Yaskawa INFORM job: R2_W24(KAMERA)(-90,90)-OKAW!!.JBI

/JOB
//NAME R2_W24(KAMERA)(-90,90)-OKAW!!
///FOLDERNAME MP_TEST
//POS
///NPOS 54,54,0,5,0,0
///TOOL 0
///POSTYPE PULSE
///PULSE
C00000=123600,-12860,-54312,-41640,88148,80397
C00001=123600,-12860,-54312,-41640,88148,80397
C00002=120727,72264,45486,-43419,68187,78537
C00003=120730,72194,45402,-43416,68199,78533
C00004=120680,125282,114040,-48791,57564,83971
C00005=120680,105365,87155,-46138,61919,81546
C00006=120233,105377,87170,-46014,61686,81428
C00007=120680,105365,87155,-46138,61919,81546
C00008=120680,106282,89568,-46525,61204,81923
C00009=120680,105365,87155,-46138,61919,81546
C00010=120680,105137,86855,-46113,61967,81521
C00011=120680,105137,86855,-46113,61967,81521
C00012=120680,105137,86855,-46113,61967,81521
C00013=120282,105147,86868,-46001,61759,81415
C00014=120680,105137,86855,-46113,61967,81521
C00015=120680,105947,89012,-46459,61327,81858
C00016=120680,105137,86855,-46113,61967,81521
C00017=126632,103319,76893,-46095,68710,81214
C00018=105628,110861,70631,9181,76248,77143
C00019=90079,103598,72277,44137,82752,76276
C00020=94241,81988,53921,45576,81194,77750
C00021=94241,81988,53921,45576,81194,77750
C00022=94870,80971,52672,45434,81052,77981
C00023=94241,81988,53921,45576,81194,77750
C00024=94241,82066,55088,45641,80710,77527
C00025=94241,81988,53921,45576,81194,77750
C00026=90439,80786,48344,46103,85116,77771
C00027=91144,88736,58191,46078,83363,77287
C00028=93989,78186,49515,45558,81861,77938
C00029=93989,78186,49515,45558,81861,77938
C00030=94486,77409,48575,45448,81739,78115
C00031=93989,78186,49515,45558,81861,77938
C00032=93989,78219,50499,45608,81441,77746
C00033=93989,78186,49515,45558,81861,77938
C00034=89014,87596,51414,46328,86969,77970
C00035=117044,71985,11723,-22209,90241,74173
C00036=120735,72113,44062,-43216,68780,78274
C00037=121402,72146,45355,-43635,68530,78708
C00038=124662,56949,12200,-42482,79430,75485
C00039=120367,52960,24213,-42516,70372,77401
C00040=120494,108785,92194,-46600,60881,81998
C00041=120821,102740,83763,-45903,62519,81314
C00042=122365,100198,76797,-45341,65431,80657
C00043=120730,72194,45403,-43416,68199,78533
C00044=107638,83716,21915,3272,91251,77584
C00045=122737,105379,80503,39421,63908,84000
C00046=124412,110163,91084,40204,59985,83172
C00047=120735,72112,44061,-43216,68781,78273
C00048=121402,72146,45354,-43635,68530,78708
C00049=124480,110073,90880,40152,60017,83221
C00050=124522,108531,89026,40010,60267,83350
C00051=123404,106925,84118,39642,62487,83737
C00052=116116,74146,21472,33448,73223,88073
C00053=116116,87806,16032,32344,82007,90677
BC00000=160885,285292,992696
BC00001=160885,285292,992696
BC00002=159740,272384,1010808
BC00003=159782,272389,903274
BC00004=165429,271706,884467
BC00005=165429,264224,884467
BC00006=165429,264224,884467
BC00007=165429,264224,884467
BC00008=165429,264224,884467
BC00009=165429,264224,884467
BC00010=148950,189766,914170
BC00011=165429,189766,884467
BC00012=165429,189766,884467
BC00013=165429,189766,884467
BC00014=165429,189766,884467
BC00015=165429,189766,884467
BC00016=165429,189766,884467
BC00017=165429,189766,884467
BC00018=165429,189766,884467
BC00019=165429,165645,884467
BC00020=165429,165645,884467
BC00021=165429,165645,884467
BC00022=165429,165645,884467
BC00023=165429,165645,884467
BC00024=165429,165645,884467
BC00025=165429,165645,884467
BC00026=165429,165645,884467
BC00027=165429,230278,884467
BC00028=165429,230278,884467
BC00029=165429,230278,884467
BC00030=165429,230278,884467
BC00031=165429,230278,884467
BC00032=165429,230278,884467
BC00033=165429,230278,884467
BC00034=165429,230278,884467
BC00035=166074,230142,881925
BC00036=167687,271433,876944
BC00037=167687,271433,876944
BC00038=166263,230102,881180
BC00039=166263,230102,881180
BC00040=166263,230102,881180
BC00041=167434,171755,876574
BC00042=167434,171755,876574
BC00043=159528,215497,902904
BC00044=167434,242986,876574
BC00045=273098,271706,884467
BC00046=273098,271706,884467
BC00047=167961,332876,877344
BC00048=167961,332876,877344
BC00049=273098,231841,884467
BC00050=273098,175866,884467
BC00051=273098,175866,884467
BC00052=273098,218083,884467
BC00053=273098,304310,884467
///POSTYPE BASE
///RECTAN
///RCONF 0,0,0,0,0,0,0,0,0,0,0,0,0,0,0,0,0,0,0,0,0,0,0,0
P00006=0.222,-3.123,-1.508,0.0000,0.0000,0.0000
P00021=-0.225,-6.128,-0.405,0.0000,0.0000,0.0000
P00022=0.222,-3.123,-1.508,0.0000,0.0000,0.0000
P00023=0.143,-0.036,0.682,0.0000,0.0000,0.0000
P00024=0.145,-0.552,1.326,0.0000,0.0000,0.0000
//INST
///DATE 2023/11/22 15:59
///ATTR SC,RW
///GROUP1 RB1,BS1
NOP
'r2_W24(kamera)(-90,90)
'Path W790
SFTOF
MOVJ C00000 BC00000 VJ=20.00
CALL JOB:CLEAN-R1_LONG
MOVJ C00001 BC00001 VJ=20.00
MOVJ C00002 BC00002 VJ=20.00
MOVJ C00003 BC00003 VJ=20.00
MOVJ C00004 BC00004 VJ=20.00
MOVL C00005 BC00005 V=60.0
REFP 3 C00006 BC00006
CALL JOB:SEARCH-R1
SET P021 P006
SFTON P021
MOVL C00007 BC00007 V=60.0
REFP 3 C00008 BC00008
CALL JOB:SEARCH-R1
SET P021 P006
SFTON P021
MOVL C00009 BC00009 V=60.0
MOVJ C00010 BC00010 VJ=20.00
MOVJ C00011 BC00011 VJ=20.00
MOVL C00012 BC00012 V=60.0
REFP 3 C00013 BC00013
CALL JOB:SEARCH-R1
SET P022 P006
SFTON P022
MOVL C00014 BC00014 V=60.0
REFP 3 C00015 BC00015
CALL JOB:SEARCH-R1
SET P022 P006
SFTON P022
MOVL C00016 BC00016 V=60.0
MOVJ C00017 BC00017 VJ=20.00
MOVJ C00018 BC00018 VJ=20.00
MOVJ C00019 BC00019 VJ=20.00
MOVJ C00020 BC00020 VJ=20.00
MOVL C00021 BC00021 V=60.0
REFP 3 C00022 BC00022
CALL JOB:SEARCH-R1
SET P023 P006
SFTON P023
MOVL C00023 BC00023 V=60.0
REFP 3 C00024 BC00024
CALL JOB:SEARCH-R1
SET P023 P006
SFTON P023
MOVL C00025 BC00025 V=60.0
MOVJ C00026 BC00026 VJ=20.00
MOVJ C00027 BC00027 VJ=20.00
MOVJ C00028 BC00028 VJ=20.00
MOVL C00029 BC00029 V=60.0
REFP 3 C00030 BC00030
CALL JOB:SEARCH-R1
SET P024 P006
SFTON P024
MOVL C00031 BC00031 V=60.0
REFP 3 C00032 BC00032
CALL JOB:SEARCH-R1
SET P024 P006
SFTON P024
MOVL C00033 BC00033 V=60.0
MOVJ C00034 BC00034 VJ=20.00
MOVJ C00035 BC00035 VJ=20.00
REFP 1 C00036 BC00036
REFP 2 C00037 BC00037
MOVJ C00038 BC00038 VJ=20.00
SFTON P021
MOVJ C00039 BC00039 VJ=20.00
MACRO1 MJ#(0) ARGF9
ARCON
SFTON P022
MOVL C00040 BC00040 V=11.0
MOVL C00041 BC00041 V=10.8
ARCOF
SFTOF
MOVL C00042 BC00042 V=100.0
MOVL C00043 BC00043 V=100.0
MOVJ C00044 BC00044 VJ=20.00
MOVJ C00045 BC00045 VJ=20.00
SFTON P024
MOVL C00046 BC00046 V=100.0 PL=0
REFP 1 C00047 BC00047
REFP 2 C00048 BC00048
MACRO1 MJ#(0) ARGF9
ARCON
MOVL C00049 BC00049 V=10.5
SFTON P023
MOVL C00050 BC00050 V=10.5
ARCOF
SFTOF
MOVL C00051 BC00051 V=100.0
MOVL C00052 BC00052 V=100.0
MOVJ C00053 BC00053 VJ=20.00
DOUT OG#(200) 15
END
